FUNCTION CheckBounds : DINT
VAR_INPUT
	index, lower, upper: DINT;
END_VAR

{noflow}

IF  index < lower THEN
	CheckBounds := lower;
	oaksGVL.udiCheckBounds := oaksGVL.udiCheckBounds + 1;
ELSIF  index > upper THEN
	CheckBounds := upper;
	oaksGVL.udiCheckBounds := oaksGVL.udiCheckBounds + 1;
ELSE  
	CheckBounds := index;
END_IF
{flow}

END_FUNCTION

(* stored: Version 1.1.0.1, ProductVersion 3.1.4022.18
   POU CheckBounds: Id {4c8c0f24-d2b7-4a31-8f4c-5702f3088314}, SpecialFunc CheckBounds *)
